// TwinCAT 3 PLC project PLCSim
// ProgramVersion: 3.1.4022.3
// libraries:
//   Tc2_Standard, * (Beckhoff Automation GmbH)
//   Tc2_System, * (Beckhoff Automation GmbH)
//   Tc3_Module, * (Beckhoff Automation GmbH)
//   VisuSymbols,3.5.10.0,System
// project tree:
//   / GlobalTextList.TcGTLO, PlcTask.TcTTO, Visualization Manager.TcVMO (not stored)
//   GVLs/ GVL.TcGVL
//   POUs/ MAIN.TcPOU, Motor.TcPOU, Process.TcPOU
//   VISUs/ ElevatorSimulator.TcVIS
//   VISUs/Visualization Resources/ Elevator.TcVIS, Elevator_Pause.TcVIS
// real-time tasks:
//   TASK PlcTask: cycle T#20ms, priority 20, ADS port 350
// variable links:
//   PLCSim/PLCSim Instance <-> PLCStudent/PLCStudent Instance
//     PlcTask Inputs/GVL.iiDisplayElevat <-> PlcTask Outputs/GVL.qiDispElevat
//     PlcTask Inputs/GVL.ixDoorClose <-> PlcTask Outputs/GVL.qxDoorClose
//     PlcTask Inputs/GVL.ixLampElevat1 <-> PlcTask Outputs/GVL.qxLampElevat1
//     PlcTask Inputs/GVL.ixLampElevat2 <-> PlcTask Outputs/GVL.qxLampElevat2
//     PlcTask Inputs/GVL.ixLampElevat3 <-> PlcTask Outputs/GVL.qxLampElevat3
//     PlcTask Inputs/GVL.ixLampLevel1 <-> PlcTask Outputs/GVL.qxLampLevel1
//     PlcTask Inputs/GVL.ixLampLevel2 <-> PlcTask Outputs/GVL.qxLampLevel2
//     PlcTask Inputs/GVL.ixLampLevel3 <-> PlcTask Outputs/GVL.qxLampLevel3
//     PlcTask Inputs/GVL.ixMotorDown <-> PlcTask Outputs/GVL.qxMotorDown
//     PlcTask Inputs/GVL.ixMotorUp <-> PlcTask Outputs/GVL.qxMotorUp
//     PlcTask Outputs/GVL.qxButtElevat1 <-> PlcTask Inputs/GVL.ixButtElevat1
//     PlcTask Outputs/GVL.qxButtElevat2 <-> PlcTask Inputs/GVL.ixButtElevat2
//     PlcTask Outputs/GVL.qxButtElevat3 <-> PlcTask Inputs/GVL.ixButtElevat3
//     PlcTask Outputs/GVL.qxButtGreen <-> PlcTask Inputs/GVL.ixButtGreen
//     PlcTask Outputs/GVL.qxButtLevel1 <-> PlcTask Inputs/GVL.ixButtLevel1
//     PlcTask Outputs/GVL.qxButtLevel2 <-> PlcTask Inputs/GVL.ixButtLevel2
//     PlcTask Outputs/GVL.qxButtLevel3 <-> PlcTask Inputs/GVL.ixButtLevel3
//     PlcTask Outputs/GVL.qxButtRed <-> PlcTask Inputs/GVL.ixButtRed
//     PlcTask Outputs/GVL.qxDoorClosed <-> PlcTask Inputs/GVL.ixDoorClosed
//     PlcTask Outputs/GVL.qxDoorOpen <-> PlcTask Inputs/GVL.ixDoorOpen
//     PlcTask Outputs/GVL.qxElevatLevel1 <-> PlcTask Inputs/GVL.ixElevatLevel1
//     PlcTask Outputs/GVL.qxElevatLevel2 <-> PlcTask Inputs/GVL.ixElevatLevel2
//     PlcTask Outputs/GVL.qxElevatLevel3 <-> PlcTask Inputs/GVL.ixElevatLevel3

CONFIGURATION PLCSim
    RESOURCE PLC ON TwinCAT3
        TASK PlcTask(INTERVAL := T#20ms, PRIORITY := 20);
        PROGRAM MAIN WITH PlcTask : MAIN;
    END_RESOURCE
END_CONFIGURATION

// ---- GVLs/GVL.TcGVL
{attribute 'qualified_only'}
VAR_GLOBAL
//Output from process to PLC
	qxButtLevel1		AT %Q*:	BOOL;		(* Button at level 1 *)
	qxButtLevel2		AT %Q*:	BOOL;		(* Button at level 2 *)
	qxButtLevel3		AT %Q*:	BOOL;		(* Button at level 3 *)

	qxButtElevat1		AT %Q*:	BOOL;		(* Button 1 inside elevator *)
	qxButtElevat2		AT %Q*:	BOOL;		(* Button 2 inside elevator *)
	qxButtElevat3		AT %Q*:	BOOL;		(* Button 3 inside elevator *)

	qxButtGreen 		AT %Q*:	BOOL;		(* Green button *)
	qxButtRed			AT %Q*:	BOOL:=TRUE;	(* Red button, normally closed *)

	qxElevatLevel1		AT %Q*: BOOL;		(* Sensor at level 1 for elevator presence *)
	qxElevatLevel2		AT %Q*: BOOL;		(* Sensor at level 2 for elevator presence *)
	qxElevatLevel3		AT %Q*: BOOL;		(* Sensor at level 3 for elevator presence *)

	qxDoorClosed		AT %Q*: BOOL;		(* Sensor for door closed *)
	qxDoorOpen			AT %Q*:	BOOL;		(* Sensor for door open *)

//Input to process from PLC
	ixLampLevel1		AT %I*:	BOOL;		(* Lamp at level 1*)
	ixLampLevel2		AT %I*:	BOOL;		(* Lamp at level 2*)
	ixLampLevel3		AT %I*:	BOOL;		(* Lamp at level 3*)

	ixLampElevat1	 	AT %I*:	BOOL;		(* Lamp 1 inside elevator *)
	ixLampElevat2	 	AT %I*:	BOOL;		(* Lamp 2 inside elevator *)
	ixLampElevat3	 	AT %I*:	BOOL;		(* Lamp 3 inside elevator *)

	ixMotorDown			AT %I*:	BOOL;		(* Run motor down *)
	ixMotorUp			AT %I*:	BOOL;		(* Run motor up *)

	ixDoorClose			AT %I*:	BOOL;		(* Close door and keep it closed *)
	iiDisplayElevat		AT %I*: UINT;		(* Intiger display inside elevator *)
END_VAR

// ---- POUs/MAIN.TcPOU
PROGRAM MAIN
VAR
END_VAR

Process();

END_PROGRAM

// ---- POUs/Process.TcPOU
PROGRAM Process
VAR
	fbMotor: 					Motor;		(* Function block to run the elevator *)
	xWarning:					BOOL;		(* Warning if door not closed during moves *)
	iDoorPosition: 				INT;		(* Door position *)
	xTopLimit:					BOOL;		(* Sensor for top limit *)
	xBottomLimit:				BOOL;		(* Sensor for bottom limit *)
	xMotorRunning:				BOOL;		(* Motor signal from elevator *)
	iMotorSpeed:				UINT:=1;	(* Motor speed *)
	iElevatPos: 				DINT;		(* Elevator position *)
	xDegreeOfDifficultyBasic:	BOOL:=TRUE; (* TRUE=basic, FALSE=more advanced *)
	xButtRedInv:				BOOL;		(* Red button on panel, normaly closed*)
END_VAR

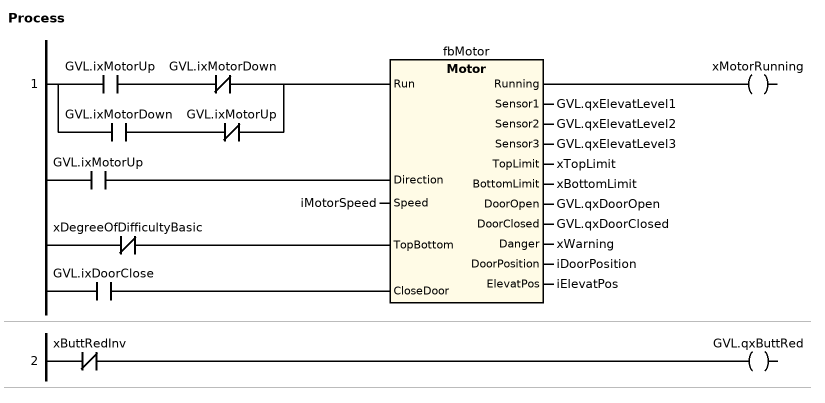
// NETWORK 1
fbMotor(
    Run := GVL.ixMotorUp AND NOT GVL.ixMotorDown OR GVL.ixMotorDown AND NOT GVL.ixMotorUp,
    Direction := GVL.ixMotorUp,
    Speed := iMotorSpeed,
    TopBottom := NOT xDegreeOfDifficultyBasic,
    CloseDoor := GVL.ixDoorClose,
    Sensor1 => GVL.qxElevatLevel1,
    Sensor2 => GVL.qxElevatLevel2,
    Sensor3 => GVL.qxElevatLevel3,
    TopLimit => xTopLimit,
    BottomLimit => xBottomLimit,
    DoorOpen => GVL.qxDoorOpen,
    DoorClosed => GVL.qxDoorClosed,
    Danger => xWarning,
    DoorPosition => iDoorPosition,
    ElevatPos => iElevatPos); // Motor
xMotorRunning := fbMotor.Running;

// NETWORK 2
GVL.qxButtRed := NOT xButtRedInv;

END_PROGRAM

// ---- POUs/Motor.TcPOU
FUNCTION_BLOCK Motor

VAR_INPUT
	Run:			BOOL;		(* Run the motor in desired direction *)
	Direction:		BOOL;		(* Direction to run in *)
	Speed:			UINT:=1;	(* Motor speed default=1 *)
	TopBottom:		BOOL;		(* If true Top and Bottom sensors are unique, if false
                               					Sensor1=Sensor1 OR Bottom; Sensor3=Sensor3 OR Top; 
                               					BottomLimit=FALSE; TopLimit=False*)
	CloseDoor: 		BOOL;		(* Close door and keep it closed *)
END_VAR
VAR_OUTPUT
	Running: 		BOOL;		(* True if the motor is running *)
	Sensor1: 		BOOL;		(* Sensor for level 1 *)
	Sensor2: 		BOOL;		(* Sensor for level 2 *)
	Sensor3: 		BOOL;		(* Sensor for level 3 *)
	TopLimit: 		BOOL;		(* Top limit switch, only used if TopBottom = TRUE *)
	BottomLimit:	BOOL;   	(* Bottom limit switch, only used if TopBottom = TRUE *)
	DoorOpen: 		BOOL;		(* Sensor for door open *)
	DoorClosed: 	BOOL;		(* Sensor for door closed *)
	Danger: 		BOOL;		(* Warning if running with not closed door *)
	DoorPosition: 	INT;		(* Door position *)
	ElevatPos: 		DINT:=5;	(* Elevator position *)
END_VAR
VAR
	OldRun: 		BOOL;
	OldDirection:	BOOL;
	DoorMove:		INT;
END_VAR
VAR CONSTANT
	TopLevel:		UINT:=450;	(* These constans defines the graphic level for each floor and the virtual sesnors *)
	GroundLevel:	UINT:=0;
	Floor1:			UINT:=5;
	Floor2:			UINT:=190;
	Floor3:			UINT:=380;
	DoorOpenPos:	INT:=0;
	DoorClosedPos: 	INT:=54;
	DoorSpeed: 		INT:=6;
END_VAR

(* FunctionBlock Motor *)
(* 2008-09-19 Fredrik Danielsson University West *)
(* 2016-01-07 BoS University West, door added *)
(* 2018-11-11 Anders N, converted to TwinCAT *)
(* v.3.1 2019-01-02 BoS, updated with new IO names and limited version for student use*)

(* By the use of oldRun we simulate a small delay when starting and
   stoping the motor. The same delay is valid for the direction. *)
IF OldRun THEN
	IF OldDirection THEN
		ElevatPos:=ElevatPos+Speed;
	ELSE
		ElevatPos:=ElevatPos-Speed;
	END_IF;

	Running:=TRUE;
ELSE
	Running:=FALSE;
END_IF;


IF ElevatPos>=TopLevel THEN
	ElevatPos:=TopLevel;
	Running:=FALSE;
	TopLimit:=TRUE;
ELSE
	TopLimit:=FALSE;
END_IF;

IF ElevatPos<=GroundLevel THEN
	ElevatPos:=GroundLevel;
	Running:=FALSE;
	BottomLimit:=TRUE;
ELSE
	BottomLimit:=FALSE;
END_IF;


IF ElevatPos>=(Floor1-Speed*2) AND ElevatPos<=(Floor1+Speed*2) THEN
	Sensor1:=TRUE;
ELSE
	Sensor1:=FALSE;
END_IF;

IF ElevatPos>=(Floor2-Speed*2) AND ElevatPos<=(Floor2+Speed*2) THEN
	Sensor2:=TRUE;
ELSE
	Sensor2:=FALSE;
END_IF;

IF ElevatPos>=(Floor3-Speed*2) AND ElevatPos<=(Floor3+Speed*2) THEN
	Sensor3:=TRUE;
ELSE
	Sensor3:=FALSE;
END_IF;


(* If the Top and Bottom limt sensors is deactivated the we hide them here *)
IF NOT TopBottom THEN
	TopLimit:=FALSE;
	BottomLimit:=FALSE;
END_IF;

OldRun:=Run;
OldDirection:=Direction;


(* Door *)
IF CloseDoor THEN
	IF DoorPosition<DoorClosedPos THEN
		
DoorMove:=DoorMove+1;
		IF DoorMove>10 THEN
			DoorMove:=0;
			DoorPosition:=DoorPosition+DoorSpeed;
		END_IF
	END_IF
ELSE
	IF DoorPosition>DoorOpenPos THEN
		DoorMove:=DoorMove+1;
		IF DoorMove>10 THEN
			DoorMove:=0;
			DoorPosition:=DoorPosition-DoorSpeed;
		END_IF
	END_IF
END_IF

IF DoorPosition<=DoorOpenPos THEN
	DoorOpen:=TRUE;
ELSE
	DoorOpen:=FALSE;
END_IF

IF DoorPosition>=DoorClosedPos THEN
	DoorClosed:=TRUE;
ELSE
	DoorClosed:=FALSE;
END_IF

(* Warning if running elevator with not closed door *)
IF Running THEN
	IF NOT DoorClosed THEN
		Danger:=TRUE;
	ELSE
		Danger:=FALSE;
	END_IF
ELSE
	Danger:=FALSE;
END_IF

END_FUNCTION_BLOCK

// ---- GlobalTextList.TcGTLO
TEXTLIST GlobalTextList
  485 = '%s'
  271 = '1'
  272 = '2'
  273 = '3'
  851 = 'BoS Jan 2016'
  829 = 'BoS Jan 2019'
  845 = 'DANGER!\nDoor not\nclosed!'
  486 = 'Door Closed'
  844 = 'Door Open'
  297 = 'Elevator'
  852 = 'Elevator_2'
  776 = 'GREEN'
  929 = 'HIT'
  849 = 'Limit'
  880 = 'RED'
  846 = 'Sensor 1'
  847 = 'Sensor 2'
  848 = 'Sensor 3'
  850 = 'University West'
  540 = 'Ver 3.1'
  603 = 'version 3.1'
END_TEXTLIST

// ---- VISUs/ElevatorSimulator.TcVIS
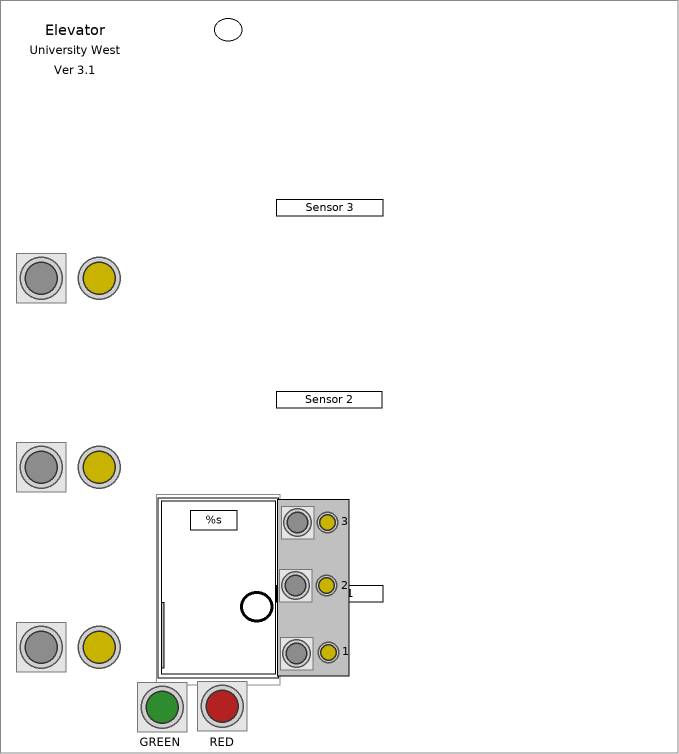
VISUALIZATION ElevatorSimulator  // 679x754
    Frame (154,497 124x191)
        shows Elevator()
        pReferences[0]: m_Input_RUNNING=Global_Variables.libMotorRunning, m_Input_LIMIT=Global_Variables.libTopLimit
        p2738717112: -Process.iElevatPos
    Frame (156,494 124x191), invisible if: true
        shows Elevator_Pause()
        p2738717112: -Process.iElevatPos
    Rectangle (30,340 100x80), "DANGER! Door not closed!"
    Rectangle (21,332 120x100), invisible if: Process.xWarning
    Rectangle (276,585 107x17), "Sensor 1", colour toggle: GVL.qxElevatLevel1
    Rectangle (276,391 106x17), "Sensor 2", colour toggle: GVL.qxElevatLevel2
    Rectangle (276,199 107x17), "Sensor 3", colour toggle: GVL.qxElevatLevel3
    Polyline (74,489)
    Polyline (266,5)
    Polyline (74,299)
    Polyline (74,109)
    Polyline (74,668)
    Polyline (142,6)
    Polyline (143,108)
    Ellipse (214,18 28x23), colour toggle: Process.xMotorRunning
    Rectangle (20,40 110x20), "University West"
    Rectangle (20,60 110x20), "Ver 3.1"
    Rectangle (161,602 3x66)
        p2738717112: -Process.iElevatPos
        p874137650: Process.iDoorPosition*2
    Rectangle (20,20 110x20), "Elevator"
    Lamp1 (74,622 50x50), variable: GVL.ixLampLevel1, style: Lamp-Lamp1-Yellow
    PushSwitch (16,622 50x50), variable: GVL.qxButtLevel1, behaviour: TAP, style: Switch-PushSwitch-Gray
    Lamp1 (74,442 50x50), variable: GVL.ixLampLevel2, style: Lamp-Lamp1-Yellow
    PushSwitch (16,442 50x50), variable: GVL.qxButtLevel2, behaviour: TAP, style: Switch-PushSwitch-Gray
    Lamp1 (74,253 50x50), variable: GVL.ixLampLevel3, style: Lamp-Lamp1-Yellow
    PushSwitch (16,253 50x50), variable: GVL.qxButtLevel3, behaviour: TAP, style: Switch-PushSwitch-Gray
    PushSwitch (137,682 50x50), variable: GVL.qxButtGreen, behaviour: TAP, style: Switch-PushSwitch-Green
    PushSwitch (197,681 50x50), variable: Process.xButtRedInv, behaviour: TAP, style: Switch-PushSwitch-Red
    Line (677,73)
    Group (277,499 79x177)
        p2738717112: -Process.iElevatPos
        Rectangle (0,0 72x177)
        Lamp1 (39,141 25x25), variable: GVL.ixLampElevat1, style: Lamp-Lamp1-Yellow
        Lamp1 (37,74 25x25), variable: GVL.ixLampElevat2, style: Lamp-Lamp1-Yellow
        Lamp1 (38,11 25x25), variable: GVL.ixLampElevat3, style: Lamp-Lamp1-Yellow
        Label (57,9 21x27), "3"
        Label (58,139 21x27), "1"
        Label (57,73 21x27), "2"
        PushSwitch (3,137 33x35), variable: GVL.qxButtElevat1, behaviour: TAP, style: Switch-PushSwitch-Gray
        PushSwitch (2,69 33x35), variable: GVL.qxButtElevat2, behaviour: TAP, style: Switch-PushSwitch-Gray
        PushSwitch (4,6 33x35), variable: GVL.qxButtElevat3, behaviour: TAP, style: Switch-PushSwitch-Gray
    Rectangle (190,510 47x20), "%s", text variable: GVL.iiDisplayElevat
        p2738717112: -Process.iElevatPos
    Rectangle (124,732 72x20), "GREEN"
    Rectangle (186,732 72x20), "RED"
END_VISUALIZATION

// ---- VISUs/Visualization Resources/Elevator.TcVIS
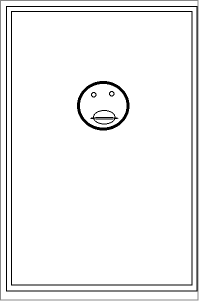
VISUALIZATION Elevator  // 199x301
    Rectangle (6,6 191x285)
    Rectangle (11,11 181x274)
    Ellipse (77,81 52x49)
    Polyline (117,230)
    Polyline (151,299)
    Polyline (81,297)
    Polyline (165,151)
    Polyline (73,152)
    Ellipse (93,110 22x14), invisible if: NOT Process.xMotorRunning
    Ellipse (91,92 5x5)
    Ellipse (109,91 5x5)
    Ellipse (90,117 28x2), invisible if: Process.xMotorRunning
END_VISUALIZATION

// ---- VISUs/Visualization Resources/Elevator_Pause.TcVIS
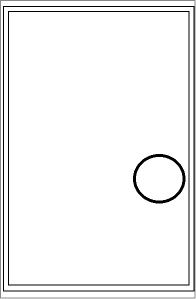
VISUALIZATION Elevator_Pause  // 196x299
    Rectangle (3,6 191x285)
    Rectangle (8,11 181x274)
    Ellipse (133,154 52x49)
    Polyline (190,297)
    Polyline (190,297)
    Polyline (119,297)
    Polyline (190,218)
    Polyline (167,217)
END_VISUALIZATION
